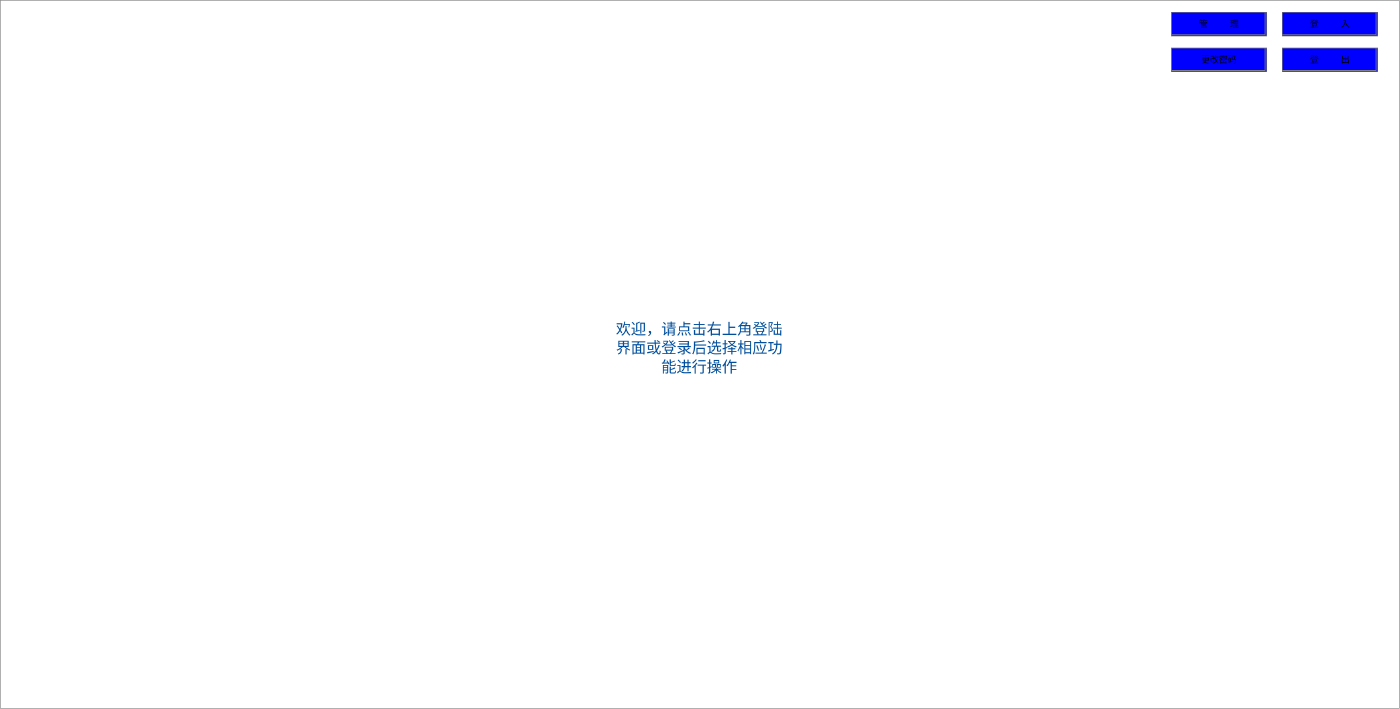
VISUALIZATION Loadding  // 1755x890, background image ImagePool1.Loadding
    Button (1607,15 120x30), "登 入"
        OnMouseClick: VisuUserMgmt Type=Login
        OnMouseClick: write the text variable via Default
    Button (1468,15 120x30), "管 理"
        OnMouseClick: VisuUserMgmt Type=OpenUserConfiguration
        OnMouseClick: write the text variable via Default
    Button (1468,60 120x30), "更改密码"
        OnMouseClick: VisuUserMgmt Type=ChangeUserPassword
        OnMouseClick: write the text variable via Default
    Button (1607,60 120x30), "登 出"
        OnMouseClick: VisuUserMgmt Type=Logout
        OnMouseClick: write the text variable via Default
        OnMouseClick: execute { VisuUserManagement.g_VisuLoginProviderManager.m_arrLoginProvider[0].stUserName:=""; }
    Rectangle (634,378 485x117), "欢迎，请点击右上角登陆 界面或登录后选择相应功 能进行操作"
END_VISUALIZATION

(* stored: Version 1.1.0.1, ProductVersion 3.1.4024.12
   Visu Loadding: Id {3d547673-01ed-43d8-85b6-a4a27b84b950} *)
